// this interface is only necessary to allow type-checking for Value Expressions
INTERFACE IValExp EXTENDS __System.IQueryInterface

END_INTERFACE

(* stored: Version 1.1.0.1
   Itf IValExp: Id {a71287c5-76cb-4acd-a801-e0e7265318c5} *)
